(* IEC 61131-3 sources: AXOpen/src/templates.simple/ax/src/templates/unit/DataManagers, 4 files *)

(* ---- FragmentsProcessDataManager.st ---- *)
NAMESPACE axosimple.UnitTemplate
    USING axosimple;
    USING AXOpen.Data;
    USING AXOpen.Core;
    USING System.Strings;

    {S7.extern=ReadWrite}
    CLASS FragmentProcessDataManger
        EXTENDS AXOpen.Data.AxoDataExchange
        VAR PUBLIC
            {#ix-generic:TOnline}
            {#ix-generic:TPlain as POCO}
            {#ix-attr:[AXOpen.Data.AxoDataEntityAttribute]}
            {#ix-attr:[Container(Layout.Stack)]}
            {#ix-set:AttributeName = "<#UnitTemplate#>"}
            Payload : axosimple.UnitTemplate.ProcessData;
        END_VAR
    END_CLASS
END_NAMESPACE

(* ---- FragmentTechnologyDataManger.st ---- *)
NAMESPACE axosimple.UnitTemplate
    USING axosimple;
    USING AXOpen.Data;
    USING AXOpen.Core;
    USING System.Strings;

    {S7.extern=ReadWrite}
    CLASS FragmentTechnologyDataManger
        EXTENDS AXOpen.Data.AxoDataExchange
        VAR PUBLIC
            {#ix-generic:TOnline}
            {#ix-generic:TPlain as POCO}
            {#ix-attr:[AXOpen.Data.AxoDataEntityAttribute]}
            {#ix-attr:[Container(Layout.Stack)]}
            {#ix-set:AttributeName = "<#UnitTemplate#>"}
            Payload : axosimple.UnitTemplate.TechnologyData;
        END_VAR
    END_CLASS
END_NAMESPACE

(* ---- ProcessDataManger.st ---- *)
NAMESPACE axosimple.UnitTemplate
    USING axosimple;
    USING AXOpen.Data;
    USING AXOpen.Core;
    USING System.Strings;

    {S7.extern=ReadWrite}
    CLASS ProcessDataManager
        EXTENDS AXOpen.Data.AxoDataFragmentExchange
        VAR PUBLIC
            {#ix-attr:[AXOpen.Data.AxoDataFragmentAttribute]}
            Shared : EntityHeaderDataManager;
            {#ix-attr:[AXOpen.Data.AxoDataFragmentAttribute]}
            DataManger : FragmentProcessDataManger;
        END_VAR
    END_CLASS
END_NAMESPACE

(* ---- TechnologyDataManager.st ---- *)
NAMESPACE axosimple.UnitTemplate
    USING axosimple;
    USING AXOpen.Data;
    USING AXOpen.Core;
    USING System.Strings;

    {S7.extern=ReadWrite}
    CLASS TechnologyDataManager
        EXTENDS AXOpen.Data.AxoDataFragmentExchange
        VAR PUBLIC
            {#ix-attr:[AXOpen.Data.AxoDataFragmentAttribute]}
            Shared : TechnologyCommonDataManager;

            {#ix-attr:[AXOpen.Data.AxoDataFragmentAttribute]}
            DataManger : FragmentTechnologyDataManger;
        END_VAR
    END_CLASS
END_NAMESPACE
